INTERFACE ITF_Serial_StandardTask

PROPERTY COUNT : INT
(*This property sets and returns the number of channels found*)
GET
END_GET
SET
END_SET
END_PROPERTY

PROPERTY CHANNELS : POINTER TO Serial_Channel
(*This property accepts the start address of the SERIAL_CHANNEL array variable*)
SET
END_SET
END_PROPERTY

METHOD PUBLIC Set_Format : Serial_FunctionResult
VAR_INPUT
	CHANNEL: INT;
	PREFIX : STRING;
	SURFIX : STRING;
END_VAR
END_METHOD

(*
	2015-06-04	:
		The method ReadString80(INT,STRING_PTR) should be used to read a string with a length of up to 80 characters long. 
*)
METHOD PUBLIC ReadString80 : Serial_FunctionResult
VAR_INPUT
	CHANNEL 			: INT;					(*The serial communication channel*)
	RECEIVED_DATA		: POINTER TO STRING;	(*The address of the variable to store the received string*)
END_VAR
END_METHOD

METHOD PUBLIC SendString80 : Serial_FunctionResult
VAR_INPUT
	CHANNEL	: INT;		(*The serial communication channel*)
	DATA	: STRING;	(*The string data to be sent to via the channel. Do not include the prefix/surfix.*)
END_VAR
END_METHOD

END_INTERFACE

(* stored: Version 1.1.0.1, ProductVersion 3.1.0.36
   Itf ITF_Serial_StandardTask: Id {89c3305b-888b-46ae-94f1-5012e4bcf520}
   Property COUNT: Id {13bd3c04-fc74-46e0-bc8f-5167c9871fa9}
   Get Get: Id {00e7a12c-8d07-4f21-a3ee-b66f9c195c1c}
   Set Set: Id {ee617baf-03aa-403e-a3b7-5725c1699aa0}
   Property CHANNELS: Id {499f437a-8256-4106-97d3-58943eb44159}
   Set Set: Id {31d57135-61d6-4f66-9355-49b5f4e272f8}
   Method Set_Format: Id {686dbd16-aa63-4931-9553-9ab5a96cce4f}
   Method ReadString80: Id {a9842072-32cf-43a5-958d-5b1821d8f772}
   Method SendString80: Id {f0fe5fe8-d753-4795-a654-3e095e47e127} *)
